// TIA Portal V20 export
// export: Created 2025-12-01T14:57:10.5084444Z, ExportSetting None, DisplayName Totally Integrated Automation Portal, DisplayVersion V20 Update 3, DisplayName TIA Portal Openness, DisplayVersion V20 Update 3, DisplayName TIA Portal Version Control Interface, DisplayVersion V20 Update 3, DisplayName STEP 7 Professional, DisplayVersion V20 Update 3, DisplayName STEP 7 Safety, DisplayVersion V20 Update 2, DisplayName WinCC Basic/Comfort/Advanced, DisplayVersion V20 Update 3, DisplayName WinCC Professional, DisplayVersion V20 Update 3, DisplayName WinCC Unified, DisplayVersion V20 Update 3
FUNCTION "FC821_OrdenesDispositivos" : Void   // FC821, LAD
TITLE = "OrdenesDispositivos" - Calcular ordenes para los dispositivos
{ S7_Optimized_Access := 'FALSE' }
AUTHOR : TRACKING
NAME : 20130301
VERSION : 3.0
// - Inicializaciones
// 
// - Bucle de Dispositivos (CCPIF- CBOX)
//   - Cierre de protocolo 
//   - Busqueda de nuevo evento recibido 
//   - Tratamiento de eventos recibidos
// 
// - Bucle de Mesas (Dispositivo)
//   - Cierre de protocolo 
//   - Busqueda de nuevo evento recibido 
//   - Tratamiento de eventos recibidos
// 
// - Bucle de Maquinas (Dispositivo)
//   - Cierre de protocolo 
//   - Busqueda de nuevo evento recibido 
//   - Tratamiento de eventos recibidos
// stored: AutoNumber false, SetENOAutomatically false
   VAR_TEMP
      RecProtocoloDispositivoMesa : "UDT_ProtocoloRecDispositivo";
      P_RecProtocolo : DWord;
      P_Temporal : DWord;
      NumeroMesa : UInt;   // Numero de Mesa Actual
   END_VAR
BEGIN

NETWORK
TITLE = Inicializaciones
// Inicializacion de variables de los DB's
/////////////////////////////////////////////////////////////////////////
// --- Inicializacion de variable de los DB's



NETWORK
TITLE = Bucle de Mesas (Dipositivos)
// - Inicializacion de variables del Dispositivo (PunteroDispo y PunteroPLC)
// - Mirar si ha cerrado el protocolo
Bucle_DispositivosMesas:NOP   0;

/////////////////////////////////////////////////////////////////////////
/////////////////////////////////////////////////////////////////////////
/////////////////////////////////////////////////////////////////////////
/////////////////////////////////////////////////////////////////////////

      L     0;  // Inicializo variable, para bucle de Mesas (Dispositivos)
      T     #NumeroMesa;

/////////////////////////////////////////////////////////////////////////
// --- Empieza el recorrido por todos los dispositivos
InicioBucle_DispositivosMesa:NOP   0;
      L     #NumeroMesa;  // Incremento en uno el numero de Mesa
      L     1;
      +I;
      T     #NumeroMesa;

/////////////////////////////////////////////////////////////////////////
// Ya he recorrido todos las Mesas (Dispositivos) ?
      L     #NumeroMesa;  // Ya estan todas las Mesas (Dispositivos)
      L     "CTE_MaxMesas";
      >I;  // Ir a Maquinas (Dispositivos)
      JC    FinalFuncion;


/////////////////////////////////////////////////////////////////////////
/// Mirar Si hay Mesa Configurada (2019 / 01 /18)
      SET;

      AN    "DB850_DefinicionMesas".Mesa[#NumeroMesa].ConfigMesa.MesaPaso;
      AN    "DB850_DefinicionMesas".Mesa[#NumeroMesa].ConfigMesa.MesaCruce;
      AN    "DB850_DefinicionMesas".Mesa[#NumeroMesa].ConfigMesa.MesaMultiplesDestinos;
      AN    "DB850_DefinicionMesas".Mesa[#NumeroMesa].ConfigMesa.MesaTL;
      JC    InicioBucle_DispositivosMesa;


/////////////////////////////////////////////////////////////////////////
// --- Recoger Datos del Dispositivo (Protocolo)
      CALL  MOVE
      ( IN  := "DB841_Recepcion".DispoMesa[#NumeroMesa].Protocolo,
        OUT := #RecProtocoloDispositivoMesa
      );

      L     P##RecProtocoloDispositivoMesa;
      T     #P_RecProtocolo;



/////////////////////////////////////////////////////////////////////////
// --- Mirar si esta cerrado el protocolo
      L     "DB831_Mesas".Mesas[#NumeroMesa].EstadoOrdenDispo;
      L     0;  // Mirar si no esta Cerrado el Protocolo ?
      <>I;  // Ir a Cerrar Protocolo de la Mesa (Dispositivo)
      JC    CerrarProtocolo_DispositivosMesa;


/////////////////////////////////////////////////////////////////////////
// Ir a Buscar Evento Nuevo para la Mesa (Dispositivo)
      JU    TratarEventosRecibidos_DispositivosMesa;



NETWORK
TITLE = Cierre del Protocolo de Mesas (Dispositivos)
// - Recoger como esta el RecepOK
// - Distribuir dependiendo del Status del Protocolo
//   - Esta en Fase 1 - Esperando que se desactive RecepOK 
//   - Esta en Fase 2 - Esperando que se active RecepOK
CerrarProtocolo_DispositivosMesa:NOP   0;

/////////////////////////////////////////////////////////////////////////
/////////////////////////////////////////////////////////////////////////
/////////////////////////////////////////////////////////////////////////
/////////////////////////////////////////////////////////////////////////
// --- Distribuir dependiendo el Status del Protocolo

      L     "DB831_Mesas".Mesas[#NumeroMesa].EstadoOrdenDispo;
      L     1;  // Mirar en que Fase esta el Protocolo?
      ==I;  // Protocolo - Esta en Fase 1
      JC    ProtocoloEnFase_01_DispositivoMesa;

// Protocolo - Esta en Fase 2
      JU    ProtocoloEnFase_02_DispositivoMesa;


/////////////////////////////////////////////////////////////////////////
/////////////////////////////////////////////////////////////////////////
// --- Fase 1 - Esperando que se Desactive RecepOK del Dispositivo
ProtocoloEnFase_01_DispositivoMesa:NOP   0;
      SET;  // DesActivado la RecepOK ?
      A     "DB840_Emision".DispoMesa[#NumeroMesa].Protocolo.RecepOK;
      JC    FinCerrarProtocolo_DispositivosMesa;


// Fase 0 - Acabado el Protocolo
      L     0;
      T     "DB831_Mesas".Mesas[#NumeroMesa].EstadoOrdenDispo;

      JU    FinCerrarProtocolo_DispositivosMesa;


/////////////////////////////////////////////////////////////////////////
/////////////////////////////////////////////////////////////////////////
// --- Fase 2 - Esperando que se active RecepOK del Dispositivo
ProtocoloEnFase_02_DispositivoMesa:NOP   0;
      SET;  // Activado la RecepOK ?
      AN    "DB840_Emision".DispoMesa[#NumeroMesa].Protocolo.RecepOK;
      JC    FinCerrarProtocolo_DispositivosMesa;


// Fase 1 - Espnierando que desactive el RecpOK
      L     1;
      T     "DB831_Mesas".Mesas[#NumeroMesa].EstadoOrdenDispo;

      L     LW [#P_RecProtocolo];
      L     W#16#80;
      AW;  // Desactivo la Orden enviada
      T     LW [#P_RecProtocolo];

      CALL  MOVE
      ( IN  := #RecProtocoloDispositivoMesa,
        OUT := "DB841_Recepcion".DispoMesa[#NumeroMesa].Protocolo
      );

      L     0;  // Borrar Words Auxiliares
      T     "DB841_Recepcion".DispoMesa[#NumeroMesa].Auxiliar_01;
      T     "DB841_Recepcion".DispoMesa[#NumeroMesa].Auxiliar_02;
      T     "DB841_Recepcion".DispoMesa[#NumeroMesa].Auxiliar_03;
      T     "DB841_Recepcion".DispoMesa[#NumeroMesa].ORDE;

      JU    FinCerrarProtocolo_DispositivosMesa;


/////////////////////////////////////////////////////////////////////////
/////////////////////////////////////////////////////////////////////////
// --- Final del Segmento del Cierre de Protocolo
FinCerrarProtocolo_DispositivosMesa:NOP   0;
// Finalizar, ir al Siguiente Dispositivo
      JU    InicioBucle_DispositivosMesa;



NETWORK
TITLE = Busqueda de nuevo evento para las Mesas (Dispositivo)
// - Pasos a seguir:
//   - Mirar si se puede tratar el evento recibido
//   - Mirar si hay algun evento recibido
//   - Distribucion de los eventos recibidos
TratarEventosRecibidos_DispositivosMesa:NOP   0;

/////////////////////////////////////////////////////////////////////////
/////////////////////////////////////////////////////////////////////////
/////////////////////////////////////////////////////////////////////////
/////////////////////////////////////////////////////////////////////////
// -- Condiciones para enviar alguna orden:
//    - StatusEmisino = 0
//    - StatusRecepcion <> 0
//

/////////////////////////////////////////////////////////////////////////
// --- Mirar si se puede Enviar orden (StatusEmision = 0)
      L     "DB831_Mesas".Mesas[#NumeroMesa].EstadoEmisionEvento;
      L     0;  // Esta emitido todo (Eventos)
      <>I;  // No se puede enviar orden
      JC    FinEventosRecibidos_DispositivosMesa;

/////////////////////////////////////////////////////////////////////////
// --- Mirar si hay algo que Enviar (StatusRecepcion <> 0)
      L     "DB831_Mesas".Mesas[#NumeroMesa].EstadoRecepcionEvento;
      L     0;  // Ha recibido algun Evento ?
      ==I;  // No Ha recibido Ninguno
      JC    FinEventosRecibidos_DispositivosMesa;


/////////////////////////////////////////////////////////////////////////
/////////////////////////////////////////////////////////////////////////
/////////////////////////////////////////////////////////////////////////
// --- Distribucion para el Tratamiento del Evento Recibido

/////////////////////////////////////////////////////////////////////////
// --- Peticion de Refresco de Datos del Dispositivo
      L     "DB831_Mesas".Mesas[#NumeroMesa].EstadoRecepcionEvento;
      L     250;
      ==I;
      JC    RefrescoDatosEventosRecibidos_DispositivosMesa;


/////////////////////////////////////////////////////////////////////////
// --- Nuevo Estado del Dispositivo >>> Sin Orden
      L     "DB831_Mesas".Mesas[#NumeroMesa].EstadoRecepcionEvento;
      L     260;
      ==I;
      JC    RefrescoDatosEventosRecibidos_DispositivosMesa;


/////////////////////////////////////////////////////////////////////////
// --- Solo queda este tipo de evento: 260...274  (Nuevo Estado del Dispositivo)
      L     "DB831_Mesas".Mesas[#NumeroMesa].EstadoRecepcionEvento;
      L     261;
      <I;  // < 260 ? - No es Nuevo Estado
      JC    DefectoEventosRecibidos_DispositivosMesa;
      L     "DB831_Mesas".Mesas[#NumeroMesa].EstadoRecepcionEvento;
      L     274;
      >I;  // > 274 ? - No es Nuevo Estado
      JC    DefectoEventosRecibidos_DispositivosMesa;

/////////////////////////////////////////////////////////////////////////
// Si es Nuevo Estado
      JU    NuevoEstadoEventosRecibidos_DispositivosMesa;


/////////////////////////////////////////////////////////////////////////
/////////////////////////////////////////////////////////////////////////
/////////////////////////////////////////////////////////////////////////
// --- Dar por tratada, no esta programado este Evento recibido
DefectoEventosRecibidos_DispositivosMesa:NOP   0;
      L     0;  // Darlo por tratado
      T     "DB831_Mesas".Mesas[#NumeroMesa].EstadoRecepcionEvento;

      JU    FinEventosRecibidos_DispositivosMesa;


/////////////////////////////////////////////////////////////////////////
/////////////////////////////////////////////////////////////////////////
/////////////////////////////////////////////////////////////////////////
// --- Final del Segmento de Buscar Nuevo Evento
FinEventosRecibidos_DispositivosMesa:NOP   0;
// Finalizar, ir al Siguiente Dispositivo
      JU    InicioBucle_DispositivosMesa;



NETWORK
TITLE = Tratamiento de los eventos para las Mesas (Dispositivos)
// - Lista de Eventos Recibidos
//   - Evento de Peticion de Refresco de datos
//   - Evento de Nuevo Estado
/////////////////////////////////////////////////////////////////////////
/////////////////////////////////////////////////////////////////////////
/////////////////////////////////////////////////////////////////////////
// --- Evento de Peticion de Refresco de Datos del Dispositivo
//     * Mirar si EstadoGeneral esta libre
//     * Darlo por tratado
//       Activacion de Generacion del Evento de Peticion de Refresco
RefrescoDatosEventosRecibidos_DispositivosMesa:NOP   0;
      L     "DB831_Mesas".Mesas[#NumeroMesa].EstadoGeneralEvento;
      L     0;  // EstadoGeneral - Libre
      <>I;
      JC    FinEventosRecibidos_DispositivosMesa;

/////////////////////////////////////////////////////////////////////////
// --- Darlo por tratado y Activacion de Generacion de Evento
      L     25;  // 25 - Refresco de Datos del dispositivo
      T     "DB831_Mesas".Mesas[#NumeroMesa].EstadoGeneralEvento;
      L     0;  // Darlo por tratado
      T     "DB831_Mesas".Mesas[#NumeroMesa].EstadoRecepcionEvento;

/////////////////////////////////////////////////////////////////////////
// --- Fin Evento de Peticion de Refresco de Datos del Dispositivo
      JU    FinEventosRecibidos_DispositivosMesa;


/////////////////////////////////////////////////////////////////////////
/////////////////////////////////////////////////////////////////////////
/////////////////////////////////////////////////////////////////////////
// --- Evento de Nuevo Estado del Dispositivo
//     * Calculo del Nuevo Estado Recibido
//     * Activar Nuevo Estado
//     * Darlo por tratado este Evento
//       Activar Protocolo del Dispositivo

/////////////////////////////////////////////////////////////////////////
// --- Calcula del Nuevo Estado Recibido
NuevoEstadoEventosRecibidos_DispositivosMesa:NOP   0;
      L     "DB831_Mesas".Mesas[#NumeroMesa].EstadoRecepcionEvento;
      L     260;
      -I;  // Numero de Bit a Activar
      L     #P_RecProtocolo;
      +D;  // Direccion del Bit a Activar
      T     #P_Temporal;

/////////////////////////////////////////////////////////////////////////
// --- Activar Orden Recibida (Nuevo Estado)

      SET;  // Poner a '1' el bit de la orden
      S     L [#P_Temporal];  // Orden del PLC calculada

      CALL  MOVE
      ( IN  := #RecProtocoloDispositivoMesa,
        OUT := "DB841_Recepcion".DispoMesa[#NumeroMesa].Protocolo
      );

/////////////////////////////////////////////////////////////////////////
// --- Darlo por tratado y Activar Protocolo
      L     2;  // Fase 2 - Esperando que active el RecepOK
      T     "DB831_Mesas".Mesas[#NumeroMesa].EstadoOrdenDispo;
      L     0;  // Darlo por tratado
      T     "DB831_Mesas".Mesas[#NumeroMesa].EstadoRecepcionEvento;


/////////////////////////////////////////////////////////////////////////
// --- Fin Evento de Nuevo Estado del Dispositivo
      JU    FinEventosRecibidos_DispositivosMesa;



NETWORK
TITLE = Final de la funcion
// Se acabo
FinalFuncion:NOP   0;

END_FUNCTION
